{attribute 'qualified_only'}
VAR_GLOBAL
	currentRowNum:UINT;
	currentStepNum:UINT;
END_VAR

(* stored: Version 1.1.0.1, ProductVersion 3.1.4024.11
   GVL AutoRowsVisu: Id {0299db4e-e4bc-0255-0cfa-c594b9793cd5} *)
